// TIA Portal V19 export
DATA_BLOCK "Liquid_Pump"   // DB10
// stored: InstanceOfName VFD Type, InstanceOfType FB
"VFD Type"
   // VAR_INPUT
   //    Overload_IN { ExternalAccessible := 'False'; ExternalVisible := 'False'; ExternalWritable := 'False'} : Bool;
   //    Isolator_in { ExternalAccessible := 'False'; ExternalVisible := 'False'; ExternalWritable := 'False'} : Bool;
   //    "Motor Number" : Int;
   //    HWIDSTW { ExternalAccessible := 'False'; ExternalVisible := 'False'; ExternalWritable := 'False'} : HW_IO;
   //    HWIDZSSW { ExternalAccessible := 'False'; ExternalVisible := 'False'; ExternalWritable := 'False'} : HW_IO;
   //    "POPUP NUmber" : Int;
   //    "Auto Run" : Bool;
   //    "Auto Speed" : Real;
   //    "Ack Error" : Bool;
   //    Ref_Speed { ExternalAccessible := 'False'; ExternalVisible := 'False'; ExternalWritable := 'False'} : Real;
   //    Ref_Current : Real;
   //    Ref_Torque { ExternalAccessible := 'False'; ExternalVisible := 'False'; ExternalWritable := 'False'} : Real;
   // END_VAR
   // VAR_OUTPUT
   //    "Drive Running" : Bool;
   //    "Actual Speed" : Real;
   //    Axis_Active : Bool;
   //    Lockout_Active : Bool;
   //    Error_Present : Bool;
   //    VFD_Fault : Int;
   //    "Motor State" : Int;
   //    Act_Current : Real;
   //    Act_torque : Real;
   // END_VAR
   // VAR_IN_OUT
   //    drive_status { ExternalAccessible := 'False'; ExternalVisible := 'False'; ExternalWritable := 'False'} : Word;
   // END_VAR
   // VAR
   //    Speed_SP : Real;
   //    "Sts Running" : Bool;
   // END_VAR
   // VAR RETAIN
   //    IEC_Counter_0_Instance { ExternalAccessible := 'False'; ExternalVisible := 'False'; ExternalWritable := 'False'} : CTU_INT;
   // END_VAR
   // VAR
   //    "SCALED sp" : Real;
   //    "speed to drive" : Real;
   //    Speed_From_Drive : Real;
   //    "SCALED sp_1" : Real;
   // END_VAR
BEGIN
END_DATA_BLOCK
